INTERFACE Resettable

METHOD reset : PVOID
VAR_INPUT
END_VAR
END_METHOD

END_INTERFACE

(* stored: Version 1.1.0.1, ProductVersion 3.1.4024.12
   Itf Resettable: Id {7ce53b0d-681b-4de4-bec2-f0f7371f2ffd}
   Method reset: Id {573e045f-518f-4a20-a022-a62fb9b636a0} *)
